INTERFACE I_MotionStage

METHOD AbsoluteMove
VAR_INPUT
	Position :LREAL;
	Velocity :LREAL;
	Acceleration :LREAL;
	Deceleration :LREAL;
END_VAR
END_METHOD

METHOD AbsoluteMoveWithBacklashCompensation
VAR_INPUT
	Position :LREAL;
	Velocity :LREAL;
	Acceleration :LREAL;
	Deceleration :LREAL;
END_VAR
END_METHOD

PROPERTY ExMotionStatus : REFERENCE TO ST_ExtendedMotionStatus
GET
END_GET
END_PROPERTY

METHOD Halt
VAR_INPUT
END_VAR
END_METHOD

METHOD Home
VAR_INPUT
	HomePosition	: LREAL;
	HomeMode	: INT;
END_VAR
END_METHOD

PROPERTY MotionCmd : REFERENCE TO ST_MotionCommand
GET
END_GET
END_PROPERTY

PROPERTY MotionStatus : REFERENCE TO ST_MotionStatus
GET
END_GET
END_PROPERTY

METHOD Reset
VAR_INPUT
END_VAR
END_METHOD

METHOD StateMove
VAR_INPUT
	Execute : BOOL;
END_VAR
END_METHOD

END_INTERFACE

(* stored: Version 1.1.0.1
   Itf I_MotionStage: Id {e70d39c3-0a78-4585-bccf-8dc4205f7d43}
   Method AbsoluteMove: Id {2011cf23-7904-4737-a6a0-b143c8fb9016}
   Method AbsoluteMoveWithBacklashCompensation: Id {bad890a2-475f-45aa-9b4a-15b622c26192}
   Property ExMotionStatus: Id {27f8593a-8fe9-40da-86a4-233d57089aba}
   Get Get: Id {5d029bcf-a2b0-4556-b6ff-6bafa16fd17d}
   Method Halt: Id {8f721796-f851-4eec-af96-2681a21359d1}
   Method Home: Id {c958a13c-5d38-4350-8e0b-a772cb5b80d0}
   Property MotionCmd: Id {a020c6dd-0fce-4bed-96e1-b266caf931a8}
   Get Get: Id {1202f2ab-b61e-4594-a4e4-9fb83a8ce3d0}
   Property MotionStatus: Id {db533644-c41f-4c47-bd41-694fd757a109}
   Get Get: Id {ea9ad5d8-c84f-4a08-bf7d-3777ab0e1cc9}
   Method Reset: Id {3872691d-974f-48d7-b1ec-fa1f41c3188e}
   Method StateMove: Id {c0f3b55a-12cb-4b52-9910-d9422a92c5c0} *)
